{attribute addProperty BoxType "EK1100-0000-0018"}
{attribute addProperty Id "Beckhoff_AX86xxEK1122Beckhoff_AX86xxEK1122_703235806352794"}
{attribute addProperty CRC "2317286561"}
{attribute addProperty SizeInBites "6352"}
{attribute addProperty SizeInBytes "794"}
TYPE Beckhoff_AX86xx_8A1EFCA1 EXTENDS EK1100_179A0949 :
STRUCT
	{attribute addProperty Name "Beckhoff_AX86xxEK1122"}
	Beckhoff_AX86xxEK1122 : Beckhoff_AX86xxEK1122_70323580;
END_STRUCT
END_TYPE

(* stored: Version 1.2.0.0, ProductVersion 3.1.4024.9
   DUT Beckhoff_AX86xx_8A1EFCA1: Id {4592397d-2800-4360-a47b-f3383a9937ff} *)
